TYPE E_ContactorFault :
(
    NONE := 0,          // Arıza yok
    FEEDBACK := 1,      // Geri besleme hatası
    WELDED := 2,        // Kontak yapışması
    COIL := 3           // Bobin arızası
);
END_TYPE

(* stored: Version 1.1.0.1, ProductVersion 3.1.4024.15
   EnumerationTextList E_ContactorFault: Id {39449036-9933-43b0-a827-9b0ecdd39be9} *)
